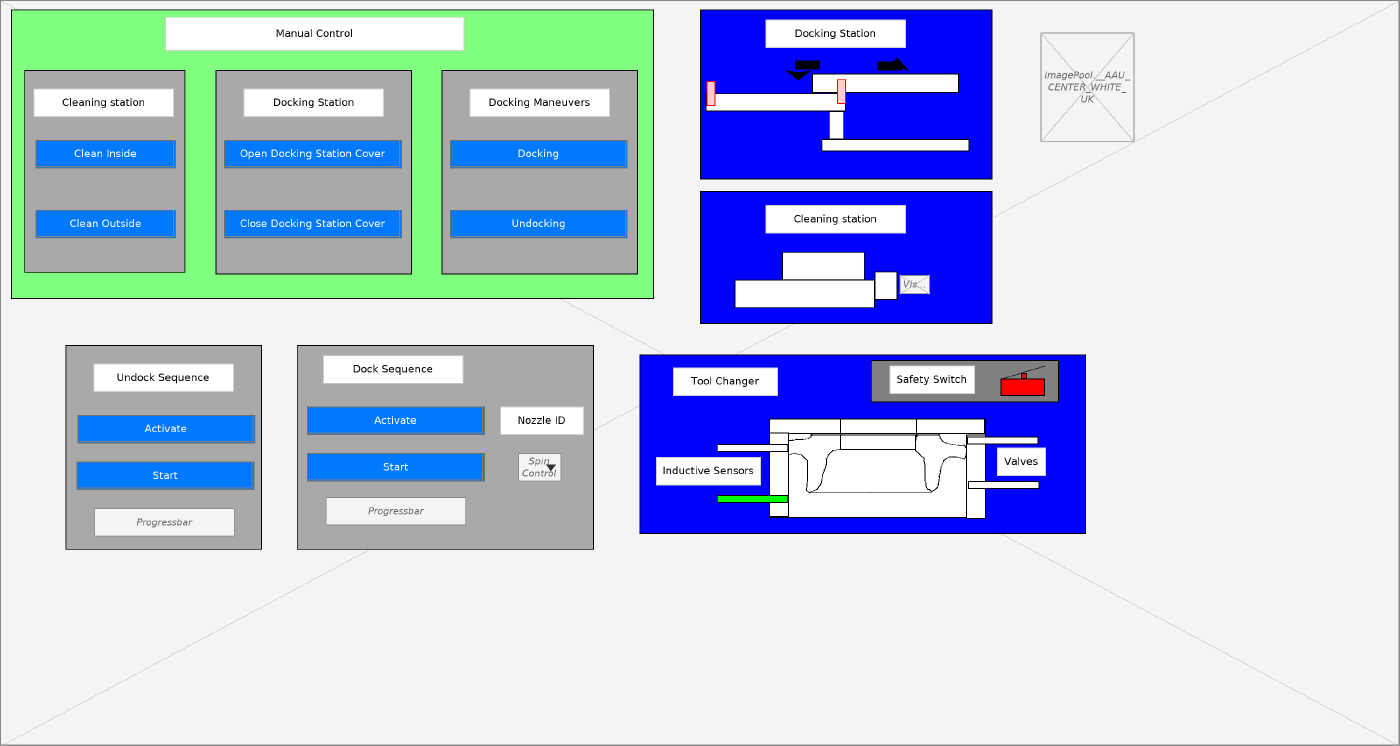
VISUALIZATION Visualization  // 1500x800
    Image (0,0 1500x800), image: ImagePool.Lasercut
    RoundedRectangle (685,380 478x192)
    RoundedRectangle (750,205 313x142)
    RoundedRectangle (750,10 313x182)
    RoundedRectangle (12,10 688x310)
    RoundedRectangle (231,75 210x219)
    RoundedRectangle (26,75 172x217)
    Button (38,150 150x30), "Clean Inside", colour toggle: CLEANout.inValve
        OnMouseClick: toggle engage.cleanIn
    Button (38,225 150x30), "Clean Outside", colour toggle: CLEANout.outValve
        OnMouseClick: toggle engage.cleanOut
    Button (240,150 190x30), "Open Docking Station Cover", colour toggle: engage.stepopen
        OnMouseClick: toggle engage.stepopen
        OnMouseClick: toggle engage.stepper
    Button (240,225 190x30), "Close Docking Station Cover", colour toggle: engage.stepclose
        OnMouseClick: toggle engage.stepclose
        OnMouseClick: toggle engage.stepper
    Textfield (36,95 150x30), "Cleaning station"
    Textfield (261,95 150x30), "Docking Station"
    RoundedRectangle (473,75 210x219)
    Button (482,150 190x30), "Docking", colour toggle: engage.dock
        OnMouseClick: toggle engage.dock
    Button (482,225 190x30), "Undocking", colour toggle: engage.undock
        OnMouseClick: toggle engage.undock
    Textfield (503,95 150x30), "Docking Maneuvers"
    RoundedRectangle (70,370 210x219)
    Button (83,445 190x30), "Activate", colour toggle: engage.allundock
        OnMouseClick: toggle engage.allundock
    Button (82,495 190x30), "Start", colour toggle: Allengage.cleanOutu
        OnMouseClick: toggle Allengage.cleanOutu
    Textfield (100,390 150x30), "Undock Sequence"
    Progressbar (101,545 150x30), variable: MAIN.allundock.step
    Textfield (177,18 320x36), "Manual Control"
    Rectangle (870,79 157x20), colour toggle: cntrlstate.cover_moving
    Rectangle (756,100 150x19)
    Rectangle (888,119 16x30)
    Rectangle (880,149 158x13)
    Textfield (820,21 150x30), "Docking Station"
    Rectangle (787,300 150x30)
    RoundedRectangle (838,270 88x30), colour toggle: cleanout.inValve
    Rectangle (937,291 24x30), colour toggle: cleanout.outValve
    Image (964,295 32x20), colour toggle: cleanout.outValve, image: VisuSymbols.Symbols.ArrowBoldRight
    Textfield (820,220 150x30), "Cleaning station"
    Rectangle (824,449 232x106)
    Rectangle (824,449 231x16)
    Group (843,465 193x63), colour toggle: cntrlstate.piston_moving
        Polyline (25,1) (58,1) (57,17) (49,18) (44,23) (42,27) (42,33) (40,39) (38,44) (36,54) (32,60) (24,63) (21,61) (22,49) (22,37) (22,29) (16,23) (11,22) (8,21) (2,23) (0,15) (2,7) (6,7) (10,6) (17,6) (23,5) (26,3) (27,0)
        Polyline (135,1) (163,1) (164,5) (167,8) (171,10) (184,12) (190,12) (193,17) (192,22) (190,27) (182,25) (174,25) (170,27) (168,29) (165,35) (164,40) (163,46) (162,54) (161,58) (160,59) (157,61) (155,62) (153,60) (151,60) (149,57) (149,53) (148,51) (148,47) (148,43) (148,38) (148,37) (148,34) (147,29)
        Polyline (147,30) (147,26) (144,24) (142,22) (138,18) (138,10) (139,0) (139,3)
        Rectangle (57,1 81x16)
        Line (24,63) (155,62)
    Rectangle (824,464 21x90)
    Rectangle (1035,466 21x90)
    Rectangle (768,476 76x8), colour toggle: TCin.ProxUp
    Rectangle (768,531 76x8), colour toggle: TCin.ProxUp
    Textfield (703,490 112x30), "Inductive Sensors"
    Rectangle (757,87 9x26), colour toggle: DSin.endStopBck
    Rectangle (897,85 9x26), colour toggle: DSin.endStopFrnt
    Textfield (721,394 112x30), "Tool Changer"
    Rectangle (1036,468 76x8), colour toggle: TCout.valvepush
    Rectangle (1037,516 76x8), colour toggle: TCout.valvepull
    Textfield (1068,480 52x30), "Valves"
    RoundedRectangle (318,370 318x219)
    Button (329,436 190x30), "Activate", colour toggle: engage.alldock
        OnMouseClick: toggle engage.alldock
    Button (329,486 190x30), "Start", colour toggle: Allengage.cleanOutd
        OnMouseClick: toggle Allengage.cleanOutd
    Textfield (346,381 150x30), "Dock Sequence"
    Progressbar (349,533 150x30), variable: MAIN.alldock.step
    SpinControl (555,486 46x30), variable: DSin.ID
        tap DSin.ID
    Textfield (536,436 89x30), "Nozzle ID"
    RoundedRectangle (933,386 201x45)
    Rectangle (1072,406 47x18), colour toggle: TCin.CollisionSW
    RoundedRectangle (1094,400 6x6), colour toggle: MAIN.switchclk.swXgood
    Line (1073,406) (1119,392)
    Textfield (953,392 91x30), "Safety Switch"
    Rectangle (940,66 26x9), colour toggle: engage.stepclose
    Polygon (946,76) (961,62) (974,76) (962,72) (956,72), colour toggle: engage.stepclose
    Rectangle (852,65 26x9), colour toggle: engage.stepopen
    Polygon (841,75) (855,86) (869,75) (857,77) (855,77), colour toggle: engage.stepopen
    Rectangle (900,449 82x16)
    Image (1115,35 100x117), image: ImagePool.__AAU_CENTER_WHITE_UK
END_VISUALIZATION

(* stored: Version 1.1.0.1, ProductVersion 3.1.4024.5
   Visu Visualization: Id {28cddda1-f6df-4ebe-b2e3-576e91a1a266} *)
